Universal Robots PolyScope program: shaft_turning.urp

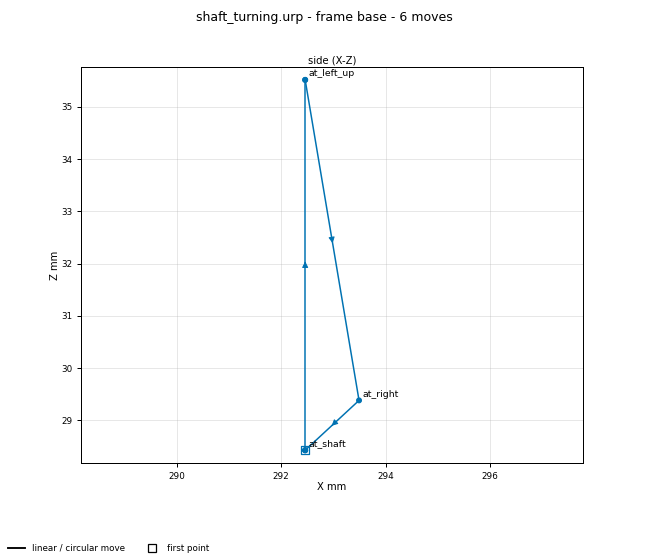
[picture p0: tool path of shaft_turning.urp in frame base, 6 of 6 moves have a stored position in this frame; points joined in program order, loops and branches not executed]
Program shaft_turning (installation=default directory=/programs/wrs2020 createdIn=5.7.0.90932 lastSavedIn=5.10.0.106288 robotSerialNumber=20205500607)
Calibrated DH parameters: a=[0.000096, -0.337, -0.383372, 0.000118, 0.000015, 0]; d=[0.162724, 79.377998, -95.545185, 16.300583, 0.099689, 0.099499]; alpha=[1.569249, 0.003272, 0.005201, 1.570041, -1.570219, 0]; deltaTheta=[0, 0.65664, 5.410619, 0.215927, -0.000001, 0]
Robot Program (runOnlyOnce=true)
  URCap Gripper (Robotiq_Grippers, Robotiq Inc.) dataModel(position=46.27450980392157, force=100.0, speed=100.0, positionInDouble=46.27450980392157, forceInDouble=100.0, speedInDouble=100.0, slaveIds=[9], blocking=true)
  MoveL speed 250 mm/s, acceleration 1200 mm/s^2 (useActiveTCP=true) feature=Base
    Waypoint at_shaft: TCP in base x=292.462 y=-172.285 z=28.427 mm, rx=-0.0168 ry=3.1097 rz=0.0286 rad; joints [124.781, -97.407, 145.354, -138.076, -87.656, 34.218] deg; TCP offset x=0 y=0 z=165 mm, rx=0 ry=0 rz=0 rad
  SuppressedNode
    Wait Sleep waitTime=1
  MoveL speed 250 mm/s, acceleration 1200 mm/s^2 (useActiveTCP=true) feature=Base
    Waypoint at_shaft_left: TCP in base x=292.462 y=-172.285 z=28.427 mm, rx=-0.0194 ry=2.7762 rz=0.0231 rad; joints [108.281, -105.484, 156.878, -147.157, -69.615, 18.58] deg
  URCap Gripper (Robotiq_Grippers, Robotiq Inc.) dataModel(position=100.0, force=0.0, speed=100.0, positionInDouble=100.0, forceInDouble=0.0, speedInDouble=100.0, slaveIds=[9], blocking=true)
  MoveL speed 250 mm/s, acceleration 1200 mm/s^2 (useActiveTCP=true) feature=Base
    Waypoint at_left_up: TCP in base x=292.462 y=-172.285 z=35.516 mm, rx=-0.0194 ry=2.7762 rz=0.0231 rad; joints [108.291, -107.329, 156.225, -144.658, -69.613, 18.577] deg
    Waypoint at_right_up: TCP in base x=292.462 y=-172.285 z=35.516 mm, rx=0.0082 ry=-2.6779 rz=-0.0282 rad; joints [139.501, -82.565, 127.092, -113.013, -105.753, 52.179] deg
    Waypoint at_right: TCP in base x=293.492 y=-172.285 z=29.381 mm, rx=0.0082 ry=-2.6779 rz=-0.0282 rad; joints [139.588, -81.714, 127.322, -114.069, -105.719, 52.27] deg
  URCap Gripper (Robotiq_Grippers, Robotiq Inc.) dataModel(position=46.27450980392157, force=100.0, speed=100.0, positionInDouble=46.27450980392157, forceInDouble=100.0, speedInDouble=100.0, slaveIds=[9], blocking=true)
  MoveL speed 250 mm/s, acceleration 1200 mm/s^2 (useActiveTCP=true) feature=Base
    Waypoint at_shaft: TCP in base x=292.462 y=-172.285 z=28.427 mm, rx=-0.0168 ry=3.1097 rz=0.0286 rad; joints [124.781, -97.407, 145.354, -138.076, -87.656, 34.218] deg
